// Mitsubishi GX Works2 project: 0630 조건 x10 누르면2   PLC: Q02/Q02H

PROGRAM MAIN
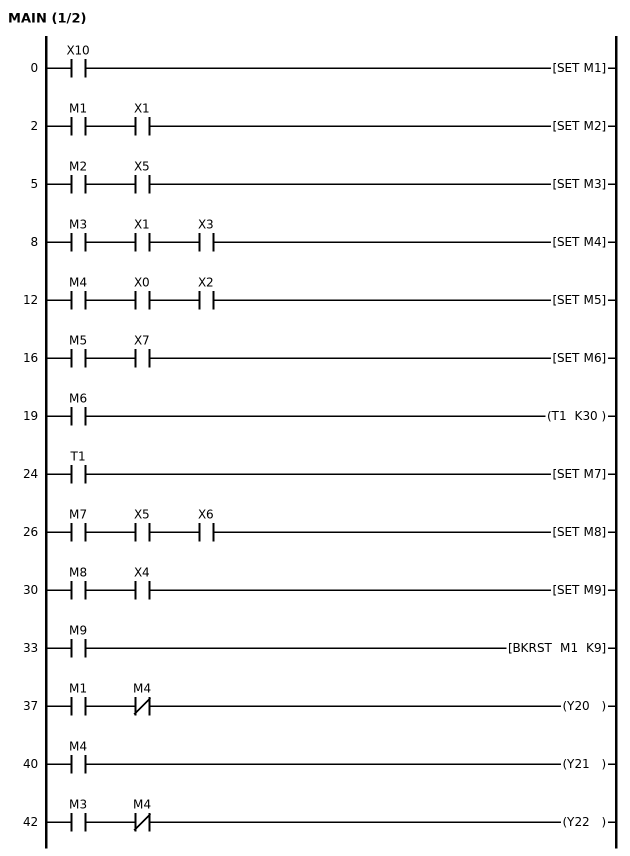
0     LD      X10
      SET     M1
2     LD      M1
      AND     X1
      SET     M2
5     LD      M2
      AND     X5
      SET     M3
8     LD      M3
      AND     X1
      AND     X3
      SET     M4
12    LD      M4
      AND     X0
      AND     X2
      SET     M5
16    LD      M5
      AND     X7
      SET     M6
19    LD      M6
      OUT     T1 K30
24    LD      T1
      SET     M7
26    LD      M7
      AND     X5
      AND     X6
      SET     M8
30    LD      M8
      AND     X4
      SET     M9
33    LD      M9
      BKRST   M1 K9
37    LD      M1
      ANI     M4
      OUT     Y20
40    LD      M4
      OUT     Y21
42    LD      M3
      ANI     M4
      OUT     Y22
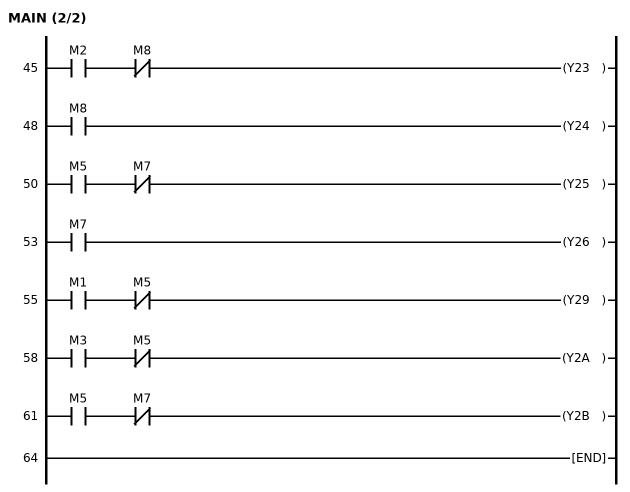
45    LD      M2
      ANI     M8
      OUT     Y23
48    LD      M8
      OUT     Y24
50    LD      M5
      ANI     M7
      OUT     Y25
53    LD      M7
      OUT     Y26
55    LD      M1
      ANI     M5
      OUT     Y29
58    LD      M3
      ANI     M5
      OUT     Y2A
61    LD      M5
      ANI     M7
      OUT     Y2B
64    END
END_PROGRAM
